Fanuc KAREL source: ka00134.KL

PROGRAM KA00134
%STACKSIZE=65535
%PRIORITY=65535
%NOLOCKGROUP
VAR
SRC : ARRAY[2] OF SHORT
DST : REAL
BEGIN
SRC[1]=2
DST=(SRC[1])
END KA00134
